PROGRAM Motor1Speed
VAR
	fbHVACMotor1Speed: FB_HVACMotor1Speed;
	eDataSecurityType: E_HVACDataSecurityType := E_HVACDataSecurityType.eHVACDataSecurityType_Idle;
	bSetDefault: BOOL;
	bEnable: BOOL;
	bAuto: BOOL;
	eCtrlModeActuator: E_HVACActuatorMode;
	bMotorProtec: BOOL;
	bFeedbContactor: BOOL;
	bFeedbProcess: BOOL;
	bRepairSwitch: BOOL;
	bManSwitch: BOOL;
	bCtrlVoltage: BOOL;
	bReset: BOOL;
	bMotor: BOOL;
	byState: BYTE;
	bStateAuto: BOOL;
	bStateRepairSwitch: BOOL;
	bStateManSwitch: BOOL;
	eStateModeActuator: Tc2_HVAC.E_HVACActuatorMode;
	bErrorGeneral: BOOL;
	byError: BYTE;
	bErrorMotorprotec: BOOL;
	bErrorFeedbContactor: BOOL;
	bErrorFeedbProcess: BOOL;
	bInvalidParameter: BOOL;
	tStartDelay: TIME;
	tStopDelay: TIME;
	tDelayFeedbContactor: TIME;
	tFeedbProcessTimer: TIME;
	tDelayFeedbProcess: TIME;
END_VAR

fbHVACMotor1Speed(
	eDataSecurityType:=eDataSecurityType, 
	bSetDefault:=bSetDefault, 
	bEnable:=bEnable, 
	bAuto:=bAuto, 
	eCtrlModeActuator:=eCtrlModeActuator, 
	bMotorProtec:=bMotorProtec, 
	bFeedbContactor:=bFeedbContactor, 
	bFeedbProcess:=bFeedbProcess, 
	bRepairSwitch:=bRepairSwitch, 
	bManSwitch:=bManSwitch, 
	bCtrlVoltage:=bCtrlVoltage, 
	bReset:=bReset, 
	bMotor=>bMotor, 
	byState=>byState, 
	bStateAuto=>bStateAuto, 
	bStateRepairSwitch=>bStateRepairSwitch, 
	bStateManSwitch=>bStateManSwitch, 
	eStateModeActuator=>eStateModeActuator, 
	bErrorGeneral=>bErrorGeneral, 
	byError=>byError, 
	bErrorMotorprotec=>bErrorMotorprotec, 
	bErrorFeedbContactor=>bErrorFeedbContactor, 
	bErrorFeedbProcess=>bErrorFeedbProcess, 
	bInvalidParameter=>bInvalidParameter, 
	tStartDelay:=tStartDelay, 
	tStopDelay:=tStopDelay, 
	tDelayFeedbContactor:=tDelayFeedbContactor, 
	tFeedbProcessTimer:=tFeedbProcessTimer, 
	tDelayFeedbProcess:=tDelayFeedbProcess);

END_PROGRAM

(* stored: Version 1.1.0.1, ProductVersion 3.1.4024.4
   POU Motor1Speed: Id {c58c5a8f-8c81-458f-bb7a-c11646322c46}, SpecialFunc None *)
